Omron CX-Programmer project NewProject (CX-Programmer 9.73)

# PLC NewPLC1: CP1E N20

## Global symbols (name address type ; comment)
0.01 BOOL  ; pb start
0.02 BOOL  ; pb stop
100.01 BOOL  ; motor
200.01 BOOL  ; relay

## Program NewProgram1 (cyclic task 0)

### Section Section1

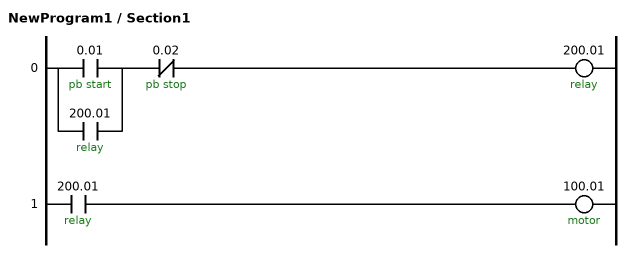
; rung 0
LD 0.01  ; pb start
OR 200.01  ; relay
ANDNOT 0.02  ; pb stop
OUT 200.01  ; relay
; rung 1
LD 200.01  ; relay
OUT 100.01  ; motor

### Section END
; rung 0
END(001)